(* IEC 61131-3 sources: Std_PalletMover/Class/_JSONReader (part 2) *)

  item := _cJSON.DetachItemFromArray(arr   :=  arr,
                                    index :=  index);

END_FUNCTION

FUNCTION GLOBAL _JSONReader::DeleteItemFromArray
	VAR_INPUT
		arr 	: ^_cJSON::t_s_cJSON;
		index 	: INT;
	END_VAR

  _cJSON.DeleteItemFromArray(arr   :=  arr,
                            index :=  index);

END_FUNCTION

FUNCTION GLOBAL _JSONReader::DetachItemFromObject
	VAR_INPUT
		parent 	: ^_cJSON::t_s_cJSON;
		item 	: ^CHAR;
	END_VAR
	VAR_OUTPUT
		retItem 	: ^_cJSON::t_s_cJSON;
	END_VAR

  retItem := _cJSON.DetachItemFromObject(parent  :=  parent,
                                        item    :=  item);

END_FUNCTION

FUNCTION GLOBAL _JSONReader::DetachItemFromObjectCaseSensitive
	VAR_INPUT
		parent 	: ^_cJSON::t_s_cJSON;
		item 	: ^CHAR;
	END_VAR
	VAR_OUTPUT
		retItem 	: ^_cJSON::t_s_cJSON;
	END_VAR

  retItem := _cJSON.DetachItemFromObjectCaseSensitive(parent  :=  parent,
                                                     item    :=  item);

END_FUNCTION

FUNCTION GLOBAL _JSONReader::DeleteItemFromObject
	VAR_INPUT
		parent 	: ^_cJSON::t_s_cJSON;
		item 	: ^CHAR;
	END_VAR

  _cJSON.DeleteItemFromObject(parent  :=  parent,
                             item    :=  item);

END_FUNCTION

FUNCTION GLOBAL _JSONReader::DeleteItemFromObjectCaseSensitive
	VAR_INPUT
		parent 	: ^_cJSON::t_s_cJSON;
		item 	: ^CHAR;
	END_VAR

  _cJSON.DeleteItemFromObjectCaseSensitive(parent  :=  parent,
                                          item    :=  item);

END_FUNCTION

FUNCTION GLOBAL _JSONReader::InsertItemInArray
	VAR_INPUT
		arr 	: ^_cJSON::t_s_cJSON;
		index 	: INT;
		newItem 	: ^_cJSON::t_s_cJSON;
	END_VAR
	VAR_OUTPUT
		result 	: BOOL;
	END_VAR

  result := _cJSON.InsertItemInArray(arr     :=  arr,
                                    index   :=  index,
                                    newItem :=  newItem);

END_FUNCTION

FUNCTION GLOBAL _JSONReader::ReplaceItemViaPointer
	VAR_INPUT
		parent 	: ^_cJSON::t_s_cJSON;
		item 	: ^_cJSON::t_s_cJSON;
		newItem 	: ^_cJSON::t_s_cJSON;
	END_VAR
	VAR_OUTPUT
		result 	: BOOL;
	END_VAR

  result := _cJSON.ReplaceItemViaPointer(parent  :=  parent,
                                        item    :=  item,
                                        newItem :=  newItem);

END_FUNCTION

FUNCTION GLOBAL _JSONReader::ReplaceItemInArray
	VAR_INPUT
		arr 	: ^_cJSON::t_s_cJSON;
		index 	: INT;
		newItem 	: ^_cJSON::t_s_cJSON;
	END_VAR
	VAR_OUTPUT
		result 	: BOOL;
	END_VAR

  result := _cJSON.ReplaceItemInArray( arr     :=  arr,
                                      index   :=  index,
                                      newItem :=  newItem);

END_FUNCTION

FUNCTION GLOBAL _JSONReader::ReplaceItemInObject
	VAR_INPUT
		object 	: ^_cJSON::t_s_cJSON;
		item 	: ^CHAR;
		newItem 	: ^_cJSON::t_s_cJSON;
	END_VAR
	VAR_OUTPUT
		result 	: BOOL;
	END_VAR

  result := _cJSON.ReplaceItemInObject(object  :=  object,
                                      item    :=  item,
                                      newItem :=  newItem);

END_FUNCTION

FUNCTION GLOBAL _JSONReader::ReplaceItemInObjectCaseSensitive
	VAR_INPUT
		object 	: ^_cJSON::t_s_cJSON;
		item 	: ^CHAR;
		newItem 	: ^_cJSON::t_s_cJSON;
	END_VAR
	VAR_OUTPUT
		result 	: BOOL;
	END_VAR

  result := _cJSON.ReplaceItemInObjectCaseSensitive( object  :=  object,
                                                    item    :=  item,
                                                    newItem :=  newItem);

END_FUNCTION

FUNCTION GLOBAL _JSONReader::Duplicate
	VAR_INPUT
		item 	: ^_cJSON::t_s_cJSON;
		recurse 	: BOOL;
	END_VAR
	VAR_OUTPUT
		retItem 	: ^_cJSON::t_s_cJSON;
	END_VAR

  retItem := _cJSON.Duplicate( item    :=  item,
                              recurse :=  recurse);

END_FUNCTION

FUNCTION GLOBAL _JSONReader::Compare
	VAR_INPUT
		compareA 	: ^_cJSON::t_s_cJSON;
		compareB 	: ^_cJSON::t_s_cJSON;
		case_sensitive 	: BOOL;
	END_VAR
	VAR_OUTPUT
		result 	: BOOL;
	END_VAR

  result := _cJSON.Compare(compareA        :=  compareA,
                          compareB        :=  compareB,
                          case_sensitive  :=  case_sensitive);

END_FUNCTION

FUNCTION GLOBAL _JSONReader::Minify
	VAR_INPUT
		json 	: ^CHAR;
	END_VAR

  _cJSON.Minify(json := json);

END_FUNCTION

FUNCTION GLOBAL _JSONReader::AddNullToObject
	VAR_INPUT
		object 	: ^_cJSON::t_s_cJSON;
		name 	: ^CHAR;
	END_VAR
	VAR_OUTPUT
		item 	: ^_cJSON::t_s_cJSON;
	END_VAR

  item := _cJSON.AddNullToObject(object  :=  object,
                                name    :=  name);

END_FUNCTION

FUNCTION GLOBAL _JSONReader::AddTrueToObject
	VAR_INPUT
		object 	: ^_cJSON::t_s_cJSON;
		name 	: ^CHAR;
	END_VAR
	VAR_OUTPUT
		item 	: ^_cJSON::t_s_cJSON;
	END_VAR

  item := _cJSON.AddTrueToObject(object  :=  object,
                                name    :=  name);

END_FUNCTION

FUNCTION GLOBAL _JSONReader::AddFalseToObject
	VAR_INPUT
		object 	: ^_cJSON::t_s_cJSON;
		name 	: ^CHAR;
	END_VAR
	VAR_OUTPUT
		item 	: ^_cJSON::t_s_cJSON;
	END_VAR

  item := _cJSON.AddFalseToObject( object  :=  object,
                                  name    :=  name);

END_FUNCTION

FUNCTION GLOBAL _JSONReader::AddBoolToObject
	VAR_INPUT
		object 	: ^_cJSON::t_s_cJSON;
		name 	: ^CHAR;
		boolean 	: BOOL;
	END_VAR
	VAR_OUTPUT
		item 	: ^_cJSON::t_s_cJSON;
	END_VAR

  item := _cJSON.AddBoolToObject(object  :=  object,
                                name    :=  name,
                                boolean :=  boolean);

END_FUNCTION

FUNCTION GLOBAL _JSONReader::AddNumberToObject
	VAR_INPUT
		object 	: ^_cJSON::t_s_cJSON;
		name 	: ^CHAR;
		number 	: LREAL;
	END_VAR
	VAR_OUTPUT
		item 	: ^_cJSON::t_s_cJSON;
	END_VAR

  item := _cJSON.AddNumberToObject(object  :=  object,
                                  name    :=  name,
                                  number  :=  number);

END_FUNCTION

FUNCTION GLOBAL _JSONReader::AddStringToObject
	VAR_INPUT
		object 	: ^_cJSON::t_s_cJSON;
		name 	: ^CHAR;
		string 	: ^CHAR;
	END_VAR
	VAR_OUTPUT
		item 	: ^_cJSON::t_s_cJSON;
	END_VAR

  item := _cJSON.AddStringToObject(object  :=  object,
                                  name    :=  name,
                                  string  :=  string);

END_FUNCTION

FUNCTION GLOBAL _JSONReader::AddRawToObject
	VAR_INPUT
		object 	: ^_cJSON::t_s_cJSON;
		name 	: ^CHAR;
		raw 	: ^CHAR;
	END_VAR
	VAR_OUTPUT
		item 	: ^_cJSON::t_s_cJSON;
	END_VAR

  item := _cJSON.AddRawToObject( object  :=  object,
                                name    :=  name,
                                raw     :=  raw);

END_FUNCTION

FUNCTION GLOBAL _JSONReader::AddObjectToObject
	VAR_INPUT
		object 	: ^_cJSON::t_s_cJSON;
		name 	: ^CHAR;
	END_VAR
	VAR_OUTPUT
		item 	: ^_cJSON::t_s_cJSON;
	END_VAR

  item := _cJSON.AddObjectToObject(object  :=  object,
                                  name    :=  name);

END_FUNCTION

FUNCTION GLOBAL _JSONReader::AddArrayToObject
	VAR_INPUT
		object 	: ^_cJSON::t_s_cJSON;
		name 	: ^CHAR;
	END_VAR
	VAR_OUTPUT
		item 	: ^_cJSON::t_s_cJSON;
	END_VAR

  item := _cJSON.AddArrayToObject( object  :=  object,
                                  name    :=  name);

END_FUNCTION

FUNCTION GLOBAL _JSONReader::SetNumber
	VAR_INPUT
		object 	: ^_cJSON::t_s_cJSON;
		number 	: LREAL;
	END_VAR
	VAR_OUTPUT
		retVal 	: LREAL;
	END_VAR

  retVal := _cJSON.SetNumber(object  :=  object,
                             number  :=  number);

END_FUNCTION

FUNCTION GLOBAL _JSONReader::SetValuestring
	VAR_INPUT
		object 	: ^_cJSON::t_s_cJSON;
		valueString 	: ^CHAR;
	END_VAR
	VAR_OUTPUT
		retVal 	: ^CHAR;
	END_VAR

  retVal := _cJSON.SetValuestring( object      :=  object,
                                   valueString :=  valueString);

END_FUNCTION

FUNCTION GLOBAL _JSONReader::ClearMainElement

  if MainElement <> NIL then
    _cJSON.Delete(item := MainElement);
  end_if;

  MainElement := NIL;

END_FUNCTION
